// TIA Portal project "Solenoid & Pilot Lamp Control with Alarm Activation" (V17)
// Solenoid & Pilot Lamp Control with Alarm Activation
// 
// PLC Example 27
// When Switch (pushbutton) is turned ON (pressed) and then turned OFF (released), then Solenoid and pilot lamp will be ON.
// And then, when Switch (pushbutton) is turned ON (pressed) and then turned OFF (released), then Solenoid and pilot lamp will be OFF and alarm will be ON.

(* hardware
DEVICE "S7-1200 station_1"  S7-1200 Station
   slot 0: "Rack_0"  S7-1200 Rack  Rack  V1.0
   slot 1: "PLC_1"  CPU 1212C AC/DC/Rly  6ES7 212-1BE40-0XB0  V4.5
*)

// ===== PLC "PLC_1"  CPU 1212C AC/DC/Rly =====

VAR_GLOBAL   // PLC tag table "Default tag table"
   "Pushbutton switch" AT %I0.0 : Bool;
   "Solenoid" AT %Q0.0 : Bool;
   "Pilot lamp" AT %Q0.1 : Bool;
   "Alarm" AT %Q0.2 : Bool;
   "Tag_1" AT %M0.0 : Bool;
   "Tag_2" AT %M0.1 : Bool;
   "Tag_3" AT %M0.2 : Bool;
END_VAR

ORGANIZATION_BLOCK "Main"   // OB1, LAD, ProgramCycle
TITLE = "Main Program Sweep (Cycle)"
{ S7_Optimized_Access := 'TRUE' }
VERSION : 0.1
   VAR_INPUT
      Initial_Call : Bool;   // Initial call of this OB
      Remanence : Bool;   // =True, if remanent data are available
   END_VAR
BEGIN

REGION Network 1
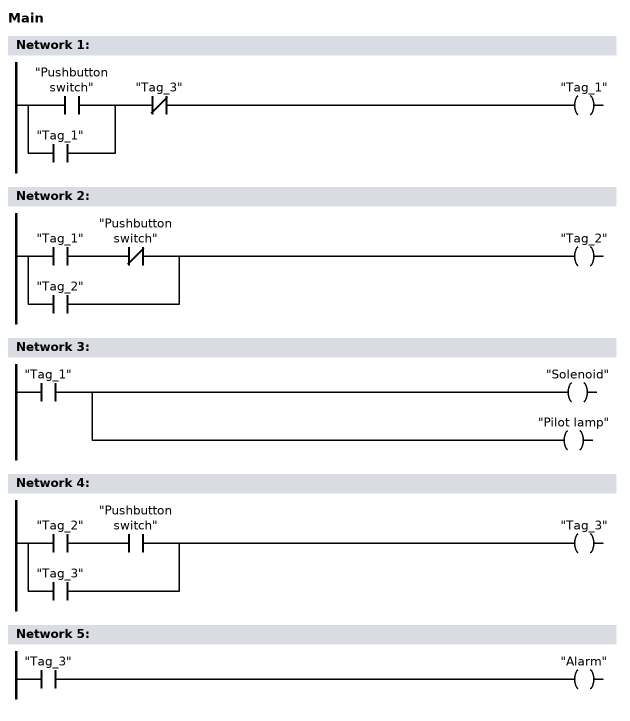
   RUNG wire#powerrail
      Contact( "Pushbutton switch" )
      wire#w1
      I_Contact( "Tag_3" )
      Coil( "Tag_1" )
   END_RUNG
   RUNG wire#powerrail
      Contact( "Tag_1" )
   END_RUNG wire#w1
   // the same network as SCL:
   "Tag_1" := ("Pushbutton switch" OR "Tag_1") AND NOT "Tag_3";
END_REGION

REGION Network 2
   RUNG wire#powerrail
      Contact( "Tag_1" )
      I_Contact( "Pushbutton switch" )
      wire#w1
      Coil( "Tag_2" )
   END_RUNG
   RUNG wire#powerrail
      Contact( "Tag_2" )
   END_RUNG wire#w1
   // the same network as SCL:
   "Tag_2" := ("Tag_1" AND NOT "Pushbutton switch") OR "Tag_2";
END_REGION

REGION Network 3
   RUNG wire#powerrail
      Contact( "Tag_1" )
      wire#w1
      Coil( "Solenoid" )
   END_RUNG
   RUNG wire#w1
      Coil( "Pilot lamp" )
   END_RUNG
   // the same network as SCL:
   "Solenoid" := "Tag_1";
   "Pilot lamp" := "Tag_1";
END_REGION

REGION Network 4
   RUNG wire#powerrail
      Contact( "Tag_2" )
      Contact( "Pushbutton switch" )
      wire#w1
      Coil( "Tag_3" )
   END_RUNG
   RUNG wire#powerrail
      Contact( "Tag_3" )
   END_RUNG wire#w1
   // the same network as SCL:
   "Tag_3" := ("Tag_2" AND "Pushbutton switch") OR "Tag_3";
END_REGION

REGION Network 5
   RUNG wire#powerrail
      Contact( "Tag_3" )
      Coil( "Alarm" )
   END_RUNG
   // the same network as SCL:
   "Alarm" := "Tag_3";
END_REGION
END_ORGANIZATION_BLOCK